FUNCTION_BLOCK FB_ADS_CAMERA EXTENDS FB_AdsBlockBase
VAR
  sAdsStruct : ST_ADS_CAMERA;
END_VAR



// Todo redirect PucPath to internal sAdsStruct instead of fb Instance
// - write InstanceName
// - or override getPucPath() (but is PRIVATE)

// The output variables are not used, please add eaccessors if needed
(*
 (*Out*)
  iO_MaxNbMarksQV           : INT := GVL_Camera.cC_QUALIVISION_MAX_NB_MARKS; 
  sO_PointsReadQV           : ST_COMMAND_PLC;    (*New points read by QualiVision*)
  iO_AvailableNbReadPointQV : INT; 
  sO_ReadPointsQV           : ARRAY[1..GVL_Camera.cC_QUALIVISION_MAX_NB_MARKS] OF ST_CAMERA_CORRECTION_QV;
*)

{attribute 'monitoring' := 'call'}
(*
  Name of the block. 
  A friendly name (which is used in the PUC to show the element (only for some blocks/apps))
*)
PROPERTY aName : T_MaxString
SET
aO_Name := aName;

sAdsStruct.aO_Name    := aO_Name;
END_SET
END_PROPERTY

PROPERTY bEnable : BOOL
GET
bEnable   := sAdsStruct.bI_Enable;   // Set ads interface variable
END_GET
SET
sAdsStruct.bI_Enable := bEnable;   // set interface variable
END_SET
END_PROPERTY

METHOD config
VAR_INPUT

END_VAR

//initRemVar();
END_METHOD

PROPERTY eCameraDevice : E_CameraDevice
GET
eCameraDevice := sAdsStruct.eI_CameraDevice;
END_GET
SET
sAdsStruct.eI_CameraDevice := eCameraDevice;
END_SET
END_PROPERTY

PROPERTY eCameraMode : E_CameraMode
GET
eCameraMode := sAdsStruct.eI_CameraMode;
END_GET
SET
sAdsStruct.eI_CameraMode := eCameraMode;
END_SET
END_PROPERTY

PROPERTY eTeachProgress : EN_CAMERA_TEACH
GET
eTeachProgress := sAdsStruct.eI_TeachProgress;
END_GET
END_PROPERTY

PROPERTY pCorrectionPointsIndication : POINTER TO ARRAY[1..4] OF ST_CORRECTION_POINT;
GET
pCorrectionPointsIndication := ADR(sAdsStruct.sI_CorrectionPointIndication);
END_GET
END_PROPERTY

PROPERTY pTeachPointsQV : POINTER TO ARRAY[1..GVL_Camera.cC_QUALIVISION_MAX_NB_MARKS] OF ST_CAMERA_TEACH_QV;
GET
pTeachPointsQV := ADR(sAdsStruct.sI_TeachPointsQV);
END_GET
END_PROPERTY

(*
  Setup constant ADS Block definitions.
  HOWTO: in abstract implmentation call
      init(aVersion:=, aType:=, nType:=, eLayer:=);
*)
METHOD  setup
init(aVersion:='01.03.00', aType:='Camera', nType:=ePr_BLK_CAMERA, eLayer:=E_AdsLayer.Structural);

// setup data in struct from init
sAdsStruct.iO_Version := iO_Version;
sAdsStruct.aO_Type    := aO_Type;
sAdsStruct.aO_Name    := aO_Name;

// redirect puc (auto-generated in base) to internal structure
_aPucPath := F_Concat2(getPucPath(), '.sAdsStruct');
END_METHOD

PROPERTY sMsgInterface : POINTER TO ST_ADS_MSG_IF
GET
sMsgInterface := ADR(sAdsStruct.sO_Message);
END_GET
END_PROPERTY

END_FUNCTION_BLOCK

(* stored: Version 1.1.0.1, ProductVersion 3.1.4024.11
   POU FB_ADS_CAMERA: Id {19330aac-119e-47f4-910c-196782e94b3a}, SpecialFunc None
   Folder Ads: Id {54730f1b-423f-4690-bea0-a250fdacbd30}
   Property aName: Id {f28f4095-3cd9-48a3-9e84-d89746b178bc}
   Set Set: Id {62382c0e-999b-4fb4-b4ee-ef61bef8a90a}
   Property bEnable: Id {b6aed005-c5f4-4179-9bb7-604707b1d09d}
   Get Get: Id {5ab39d2e-eead-4ad9-aaac-d34c08739fd8}
   Set Set: Id {ac2c63b0-1693-4ea6-9c41-8297b4eec2c4}
   Method config: Id {52de9062-328f-46bf-89b9-aa93271e499f}
   Property eCameraDevice: Id {626d17fb-0b68-4a92-8877-8e00e3ee2031}
   Get Get: Id {ad3c7d11-b19b-4c88-8d2f-40d41d3a143c}
   Set Set: Id {fd60a492-3c4e-4b92-8ebd-886106e63114}
   Property eCameraMode: Id {ee69af58-1408-4b18-bc29-7432b7433bd3}
   Get Get: Id {6700eb6b-e55b-42da-8923-08be24785fa0}
   Set Set: Id {68ccd15a-3244-4499-9912-4b98892f2354}
   Property eTeachProgress: Id {3076ebd4-2d9b-4411-9b9d-116615919886}
   Get Get: Id {aa12269c-1efb-4c47-ba8b-6c3754445d9b}
   Property pCorrectionPointsIndication: Id {25cd1b7a-7221-45a1-b906-690758f96618}
   Get Get: Id {9ad2cc44-b22a-43e5-a00c-df5b0b0a4c6a}
   Property pTeachPointsQV: Id {a3b77820-cada-437d-944c-35a78d711843}
   Get Get: Id {24c5d808-ceb3-4080-a2c4-e32c50a954a9}
   Method setup: Id {64df0548-1b08-4e9a-bf43-44acfe43b0ef}
   Property sMsgInterface: Id {01d19590-9787-42a7-9216-27c225c735f9}
   Get Get: Id {d6b10973-1e30-4177-b4c4-2ff4894a4917} *)
